// TIA Portal V19 export
DATA_BLOCK "Config"   // DB75
// stored: Access Published, MemoryReserve 100, Namespace Unit2.EM1
   VAR
      em { ExternalWritable := 'False'} : "LAF_typeEmConfiguration";   // Configuration of EM Parameters
      axis { ExternalWritable := 'False'} : Array[1.._.U2EM1_NO_OF_AXES] of DB_ANY;   // Assign the axis of the EM
      em1Parameters : "LAF_typeRollerEm1Parameters";
   END_VAR
BEGIN
   em.referenceDesignator.parent := WSTRING#'U1';
   em.referenceDesignator.relative := WSTRING#'EM1';
END_DATA_BLOCK
